{attribute 'qualified_only'}
VAR_GLOBAL
stParam		:	ST_Parameters;
END_VAR

(* stored: Version 1.1.0.1
   GVL G_Parameters: Id {bf1f20ef-581e-4190-8cbe-0310987fd2eb} *)
